(* IEC 61131-3 sources: volt/packages/volt-lsp-iec/test-corpus/pro2193/Device/Plc Logic/Application/01 Main, 4 files *)

(* ---- HardwareButtons.pou ---- *)
{attribute 'global_init_slot' := '50002'}
{attribute 'symbol' := 'none'}
PROGRAM HardwareButtons
VAR_INPUT
	StartCycle			: PushButtonWithObserverFB;
	EndCycle			: PushButtonWithObserverFB;
	Stop				: PushButtonWithObserverFB;
	Reset				: PushButtonWithObserverFB;
	Homing				: PushButtonWithObserverFB;
	F1					: PushButtonFunctionKeyFB;
	F2					: PushButtonFunctionKeyFB;
	{attribute 'symbol' := 'readwrite'}	EnableIML			: PushButtonLedWithHmiFB;
END_VAR
VAR
	startLedTest		: BOOL;
	F1OldObserverCount	: UINT;
	F2OldObserverCount	: UINT;
	speedFooterShow		: BOOL;
	SpeedFooterTimeout	: BTON;
	testestse	: BTON;
	leds				: ARRAY[1..6] OF ILed :=
	[
		StartCycle,
		EndCycle,
		Homing,
		Reset,
		F1,
		F2
	];
	leds2				: ARRAY[1..6] OF ILed :=
	[
		SER.Stacklight.Red,
		SER.Stacklight.Amber,
		SER.Stacklight.Green,
		SER.GateZAxis.ButtonUnLock,
		SER.GateZAxis.ButtonLock,
		ProcessModules.ConveyorControl.ButtonStartNewStack
	];
END_VAR
VAR CONSTANT
	speedFooterShowTime	: REAL	:= 5;	// Show footer for 5 seconds
END_VAR

%LANGUAGE ST
Initialize();

StartCycle(		buttonType		:= enumHWButtons.Start);
EndCycle(		buttonType		:= enumHWButtons.EndCycle);
Stop(			buttonType		:= enumHWButtons.Stop);
Reset(			buttonType		:= enumHWButtons.Reset);
Homing(			buttonType		:= enumHWButtons.Homing);
F1(				buttonType		:= enumHWButtons.F1);
F2(				buttonType		:= enumHWButtons.F2);
EnableIML();
LedTest();

// Switch IML on/off when hardware/software button is pushed
IF EnableIML.ButtonPushed THEN
	PersistentVars.RecipeVars.EnableIML	:= NOT PersistentVars.RecipeVars.EnableIML;
END_IF
IF NOT PersistentVars.RecipeVars.EnableIML THEN
	EnableIML.Off();
ELSIF InjectionMouldingMachine.Data.usiFirstShotsWithoutIML = 0
   OR InjectionMouldingMachine.Unit.ShotCounter > InjectionMouldingMachine.Data.usiFirstShotsWithoutIML
THEN
	EnableIML.SetColors(enumColorList.Lime);
	EnableIML.Solid();
ELSIF SER.OperationMode = SER_OperationModeType.SemiAuto THEN
	EnableIML.SetColors(enumColorList.Lime);
	EnableIML.Solid();
ELSE
	EnableIML.SetColors(enumColorList.Yellow);	// IML temporary disabled during cycle startup
	EnableIML.Solid();
END_IF

IF ErrorHandling.errorActive THEN
	Reset.Flash();
ELSE
	Reset.Off();
END_IF

GlobalVars.Reset S= Reset.ButtonPushed;
GlobalVars.Reset R= Reset.ButtonReleased;

IF F1.ObserverCount <> F1OldObserverCount THEN
	IF F1.ObserverCount > 0 THEN
		F1.Solid();
	ELSE
		F1.Off();
	END_IF
	F1OldObserverCount := F1.ObserverCount;
END_IF

IF F2.ObserverCount <> F2OldObserverCount THEN
	IF F2.ObserverCount > 0 THEN
		F2.Solid();
	ELSE
		F2.Off();
	END_IF
	F2OldObserverCount := F2.ObserverCount;
END_IF

IF SER.InAutomaticOperation
AND SER.OperationMode <> SER_OperationModeType.SemiAuto
THEN
	IF F1.ButtonPushed THEN
		PersistentVars.usiGlobalSERSpeed	:= MAX(5,	PersistentVars.usiGlobalSERSpeed - 5);
		speedFooterShow						:= TRUE;
		HMI.FooterName						:= enumFooterNames.GlobalSpeed;
		SpeedFooterTimeout.Reset();
	END_IF
	IF F2.ButtonPushed THEN
		PersistentVars.usiGlobalSERSpeed	:= MIN(100,	PersistentVars.usiGlobalSERSpeed + 5);
		speedFooterShow						:= TRUE;
		HMI.FooterName						:= enumFooterNames.GlobalSpeed;
		SpeedFooterTimeout.Reset();
	END_IF
END_IF

IF SpeedFooterTimeout.Set(In := speedFooterShow, Pt := speedFooterShowTime) THEN
	speedFooterShow		:= FALSE;
	HMI.FooterName		:= enumFooterNames.None;
END_IF

END_PROGRAM

METHOD PRIVATE Initialize
VAR_INPUT
END_VAR
VAR_INST
	{attribute 'init_on_onlchange'}
	xInitialized	: BOOL;
END_VAR

%LANGUAGE ST
IF xInitialized THEN
	RETURN;
END_IF

startLedTest := TRUE;

xInitialized := TRUE;

END_METHOD

// Do little animation with the leds during startup :)
METHOD PRIVATE LedTest
VAR_INST
	ledTestDuration		: BTON;
	ledTestStep			: BTON;
	i					: INT;
	position			: INT := 1;
END_VAR

%LANGUAGE ST
IF ledTestDuration.Set(In := startLedTest, Pt := 8) THEN
	startLedTest := FALSE;
	position := 1;
	FOR i := 1 TO 6 DO
		leds[i].LedTestStop();
		leds2[i].LedTestStop();
	END_FOR
END_IF

IF ledTestStep.Set(In := startLedTest, Pt := 0.3) THEN
	leds[SEL(position = 1, position - 1, 6)].LedTestOff();
	leds[position].LedTestOn();
	leds[SEL(position = 6, position + 1, 1)].LedTestOn();

	leds2[SEL(position = 1, position - 1, 6)].LedTestOff();
	leds2[position].LedTestOn();

	ledTestStep.Reset();
	Increment.Rollover(input := position, rollover := 6, incrementBy := 1, zeroValue := 1);
END_IF

END_METHOD

(* ---- HMI.pou ---- *)
// By default every variable here has read/write access from the HMI
{attribute 'symbol' := 'readwrite'}
PROGRAM HMI
VAR_INPUT
	xMuteHorn					: BOOL;
	OperationMode				: SER_OperationModeType;	// Unit mode change request from HMI
	FooterName					: enumFooterNames;			// Select active footer type
END_VAR
VAR_OUTPUT
	servoJogMode				: BOOL;						// False: Move to position; True: Servo jogging to sw limit.
	servoJogSpeed				: BOOL;						// False: Slow speed; True: High speed
	UUIDActiveScreen			: STRING(40);
	SemiAutoMode				: enumSemiAutoModeType;		// Choose mode when SER runs in operation mode: Semi-auto
	testMachineWithoutConveyors	: BOOL;						// Disable sensors to testrun the machine without conveyors
	currentUser					: STRING(80);				// Current user
END_VAR
VAR
	ButtonEnableDrives			: PushButtonLedWithHmiFB;
	ButtonEnableMainvalve		: PushButtonLedWithHmiFB;
	ButtonEnableVacuumPumps		: PushButtonLedWithHmiFB;
	ButtonEnableSticker			: PushButtonLedWithHmiFB;
	ButtonEnableCamera			: PushButtonLedWithHmiFB;

	{attribute 'symbol' := 'read'}	SER_State					: PACK_ML.State;
	{attribute 'symbol' := 'read'}	heartbeatToHMI				: UDINT;
	{attribute 'symbol' := 'read'}	ProjectInfo					: ProjectInfoType;
	{attribute 'symbol' := 'read'}	textMessage					: STRING(80);		// Show a custom text message as a popup on the HMI panel.
	{attribute 'symbol' := 'read'}	ipAddressController			: STRING(20);
	{attribute 'symbol' := 'read'}	ipAddressPilz				: STRING(20);
	{attribute 'symbol' := 'read'}	robotSerial					: STRING(7);		// The Serial number of the robot.

	ipAddressEdgePC				: STRING(20)	:= '10.195.0.8';
	communicationPortEdgePC		: UINT			:= 48000;
	heartbeatToPLC				: UDINT;
	logMessageParameterChange	: STRING(255);

	autoLogoffMinutes			: UINT; // Minutes of inactivity after which the current user is being logged off.

	{attribute 'init_on_onlchange'}		// Reset initialized with every online change.
	{attribute 'symbol' := 'none'}	initialized					: BOOL;
	{attribute 'symbol' := 'none'}	startGetControllerIp		: BOOL;
	{attribute 'symbol' := 'none'}	startGetRobotSerial			: BOOL;
	{attribute 'symbol' := 'none'}	heartbeatMissingAlarm		: SetErrorFB();
	{attribute 'symbol' := 'none'}	serialNumberRead			: RobotSerialNumberFB;
END_VAR
VAR CONSTANT
	{attribute 'symbol' := 'none'}	PilzAddToLastOctetOfIp		: BYTE := 2;		// IP address of Pilz PnozMulti will be 2 higher than controller IP. So controller is: 10.100.xxx.10, then Pilz is: : 10.100.xxx.12
END_VAR

%LANGUAGE ST
initialized := initialized OR_ELSE Initialize();

MonitorHeartbeat();

Cyclic();

// Get robot serial number from SD card
serialNumberRead(
	execute				:= startGetRobotSerial,
	controller			:= enumControllerType.C5xxSeries,
	busy				=> ,
	done				=> ,
	errorActive			=> ,
	errorDescription	=> ,
	robotSerial			=> );

IF serialNumberRead.done THEN
	robotSerial				:= serialNumberRead.robotSerial;
	startGetRobotSerial		:= FALSE;
END_IF

END_PROGRAM

// Get the final octet (digit) of an IP address, then increase this digit with another number
METHOD PRIVATE ChangeLastOctetOfIp : STRING(20)
VAR_INPUT
	ipAddress		: STRING(20);
	addTolastOctet	: BYTE;		// number to add to last octet
END_VAR
VAR
	index			: INT;
	lastOctet		: BYTE;
END_VAR

%LANGUAGE ST
index	:= LEN(ipAddress) - 1;	// Get index of last character in string

// Get last index of '.' (ascii: 46)
WHILE ipAddress[index] <> enumASCII.DOT AND index > 0 DO
	index := index - 1;
END_WHILE

IF index > 0 THEN
	lastOctet			:= TO_BYTE(MID(ipAddress, LEN(ipAddress) - 1 - index, index + 2)) + addTolastOctet;
	ChangeLastOctetOfIp := CONCAT(LEFT(ipAddress, index + 1), TO_STRING(lastOctet));
END_IF

END_METHOD

METHOD PRIVATE Cyclic
VAR_INST
	getControllerIp				: GetIPAddressFB;
	UUIDActiveScreenHistory		: ARRAY[0..4] OF STRING(80);
END_VAR
VAR
	i							: USINT;
END_VAR

%LANGUAGE ST
ButtonEnableDrives();
ButtonEnableMainvalve();
ButtonEnableVacuumPumps();
ButtonEnableSticker();
ButtonEnableCamera();

IF SER.xServoDrivesEnabled THEN
	ButtonEnableDrives.SetColors(enumColorList.Lime);
	ButtonEnableDrives.Solid();
ELSIF GlobalVars.EnableServoDrives THEN
	ButtonEnableDrives.SetColors(enumColorList.Blue);
	ButtonEnableDrives.Solid();
ELSE
	ButtonEnableDrives.Off();
END_IF

IF SER.DigIn.xAirPressureOK THEN
	ButtonEnableMainvalve.SetColors(enumColorList.Lime);
	ButtonEnableMainvalve.Solid();
ELSIF GlobalVars.EnableMainvalve THEN
	ButtonEnableMainvalve.SetColors(enumColorList.Blue);
	ButtonEnableMainvalve.Solid();
ELSE
	ButtonEnableMainvalve.Off();
END_IF

IF  SER.VacuumPumps.xVacuumpumpRunning
AND SER.VacuumPumps.xHighVacuumtankFull
AND (SER.VacuumPumps.xLowVacuumtankFull OR SER.VacuumPumps.xOptionDisableVacuumPump2)
THEN
	ButtonEnableVacuumPumps.SetColors(enumColorList.Lime);
	ButtonEnableVacuumPumps.Solid();
ELSIF SER.VacuumPumps.xVacuumpumpRunning THEN
	ButtonEnableVacuumPumps.SetColors(enumColorList.Blue);
	ButtonEnableVacuumPumps.Solid();
ELSE
	ButtonEnableVacuumPumps.SetColors(enumColorList.Gray);
	ButtonEnableVacuumPumps.Off();
END_IF

// Switch IML on/off when software button is pushed
IF ButtonEnableSticker.ButtonPushed AND NOT SER.InAutomaticOperation THEN
	PersistentVars.RecipeVars.EnableSticker	:= NOT PersistentVars.RecipeVars.EnableSticker;
END_IF

ButtonEnableSticker.SetColors(enumColorList.Lime);
IF PersistentVars.RecipeVars.EnableSticker THEN
	ButtonEnableSticker.Solid();
ELSE
	ButtonEnableSticker.Off();
END_IF

// Switch vision system on / off
IF ButtonEnableCamera.ButtonPushed AND NOT SER.InAutomaticOperation THEN			// by customer request only onable/disable camera when machine is off
	PersistentVars.RecipeVars.EnableVision	:= NOT PersistentVars.RecipeVars.EnableVision;
END_IF
ButtonEnableCamera.SetColors(colorOn := enumColorList.Lime);
IF PersistentVars.RecipeVars.EnableVision THEN
	ButtonEnableCamera.Solid();
ELSE
	ButtonEnableCamera.Off();
END_IF

SER_State			:= SER.ActState;

//Get ip addresses of the controller and the Pilz PnozMulti
IF startGetControllerIp THEN
	getControllerIp();
	IF getControllerIp.resultValid THEN
		ipAddressController		:= getControllerIp.currentIp;
		ipAddressPilz			:= ChangeLastOctetOfIp(ipAddressController, PilzAddToLastOctetOfIp);
		startGetControllerIp	:= FALSE;
	END_IF
END_IF

// Debugging: keep a short history of uuids
IF UUIDActiveScreen <> UUIDActiveScreenHistory[0] THEN
	FOR i := 4 TO 1 BY -1 DO
		UUIDActiveScreenHistory[i] := UUIDActiveScreenHistory[i-1];
	END_FOR
	UUIDActiveScreenHistory[0] := UUIDActiveScreen;
END_IF

END_METHOD

// Initializes the FB in the first cycle
METHOD PRIVATE Initialize : BOOL

%LANGUAGE ST
ProjectInfo				:= GetProjectInfo();
startGetControllerIp	:= TRUE;
startGetRobotSerial		:= TRUE;
Initialize				:= TRUE;

END_METHOD

METHOD PRIVATE MonitorHeartbeat
VAR_INST
	heartbeatTimer				: BTON;
	previousHeartbeat			: UDINT;
END_VAR

%LANGUAGE ST
// Send a heartbeat to the HMI every 0,5 sec. (currently not in use)
IF heartbeatTimer.Set(In := TRUE, Pt := 0.5) THEN
	heartbeatTimer.Reset();
	Increment.AnyInt(heartbeatToHMI);
END_IF

// Monitor heartbeat signal from HMI
heartbeatMissingAlarm(
	moduleHandler	:= ErrorHandling.ModuleHandler,
	textRefId		:= General_Unit_Errors,
	errorId			:= 4,		// Missing heartbeat from HMI
	alarmCondition	:= FALSE, //heartbeatToPLC = previousHeartbeat,  // Panel cannot write variables in JS loops..!
	alarmDelay		:= 5.0,
	severity		:= enumErrorSeverity.Warning,
	reaction		:= enumErrorReaction.No_reaction,
	active			=> );

previousHeartbeat := heartbeatToPLC;

// In case of a HMI crash, detach the F1 and F2 buttons from all observers by invalidating the UUID
IF heartbeatMissingAlarm.active THEN
	UUIDActiveScreen := '';
END_IF

END_METHOD

(* ---- HMI_BFU.pou ---- *)
// By default every variable here has read/write access from the HMI
{attribute 'symbol' := 'readwrite'}
// Handle the BFU specific buttons
PROGRAM HMI_BFU
VAR_INPUT
	OperationMode				: SER_OperationModeType;	// Unit mode change request from HMI
END_VAR
VAR_OUTPUT
	UUIDActiveScreen			: STRING(40);
END_VAR
VAR
	ButtonEnableDrives			: PushButtonLedWithHmiFB;
	ButtonEnableMainvalve		: PushButtonLedWithHmiFB;
	ButtonEnableVacuumPumps		: PushButtonLedWithHmiFB;

	{attribute 'symbol' := 'read'}	BFU_State					: PACK_ML.State;
END_VAR

%LANGUAGE ST
Initialize();

ButtonEnableDrives();
ButtonEnableMainvalve();
ButtonEnableVacuumPumps();

IF BFU.xServoDrivesEnabled THEN
	ButtonEnableDrives.SetColors(enumColorList.Lime);
	ButtonEnableDrives.Solid();
ELSIF GlobalVars_BFU.EnableServoDrives THEN
	ButtonEnableDrives.SetColors(enumColorList.Blue);
	ButtonEnableDrives.Solid();
ELSE
	ButtonEnableDrives.Off();
END_IF

IF BFU.DigIn.xAirPressureOK THEN
	ButtonEnableMainvalve.SetColors(enumColorList.Lime);
	ButtonEnableMainvalve.Solid();
ELSIF GlobalVars_BFU.EnableMainvalve THEN
	ButtonEnableMainvalve.SetColors(enumColorList.Blue);
	ButtonEnableMainvalve.Solid();
ELSE
	ButtonEnableMainvalve.Off();
END_IF

BFU_State			:= BFU.ActState;

END_PROGRAM

METHOD PRIVATE Initialize
VAR_INPUT
END_VAR
VAR_INST
	xInitialized	: BOOL;
END_VAR

%LANGUAGE ST
IF xInitialized THEN
	RETURN;
END_IF

xInitialized := TRUE;

END_METHOD

(* ---- Main.pou ---- *)
PROGRAM Main
VAR
	StartupTimer	: BTON;
	taskInfo				: CmpIecTask.Task_Info2;
END_VAR

%LANGUAGE ST
__TRY
taskInfo	:= TaskGetInfo();
IF NOT StartupTimer.Set(TRUE, 1) THEN	// Delay before starting program. The first PLC cycle the I/Q is not updated yet.
	IQ_Handling();
	RETURN;
END_IF

__CATCH(GVL_Exceptions.aeExceptionCodes[eExceptionCodes.MainTask])
	GVL_Exceptions.xException := TRUE;
	GVL_Exceptions.iCounter := GVL_Exceptions.iCounter + 1;
__ENDTRY

__TRY TimeSettings();		__CATCH(GVL_Exceptions.aeExceptionCodes[eExceptionCodes.TimeSettings])	GVL_Exceptions.xException := TRUE;	GVL_Exceptions.iCounter := GVL_Exceptions.iCounter + 1;		__ENDTRY		// Get or set the current date / time
__TRY EtherCAT_Diag();		__CATCH(GVL_Exceptions.aeExceptionCodes[eExceptionCodes.EtherCAT_Diag])	GVL_Exceptions.xException := TRUE;	GVL_Exceptions.iCounter := GVL_Exceptions.iCounter + 1;		__ENDTRY	// Get diagnostics about the EtherCAT connection
__TRY ErrorHandling();		__CATCH(GVL_Exceptions.aeExceptionCodes[eExceptionCodes.ErrorHandling])	GVL_Exceptions.xException := TRUE;	GVL_Exceptions.iCounter := GVL_Exceptions.iCounter + 1;		__ENDTRY
__TRY HardwareButtons();	__CATCH(GVL_Exceptions.aeExceptionCodes[eExceptionCodes.HardwareButtons])	GVL_Exceptions.xException := TRUE;	GVL_Exceptions.iCounter := GVL_Exceptions.iCounter + 1;		__ENDTRY
__TRY BfuButtons();			__CATCH(GVL_Exceptions.aeExceptionCodes[eExceptionCodes.BfuButtons])	GVL_Exceptions.xException := TRUE;	GVL_Exceptions.iCounter := GVL_Exceptions.iCounter + 1;		__ENDTRY
__TRY HMI();				__CATCH(GVL_Exceptions.aeExceptionCodes[eExceptionCodes.HMI])	GVL_Exceptions.xException := TRUE;	GVL_Exceptions.iCounter := GVL_Exceptions.iCounter + 1;		__ENDTRY		// Setup communication with HMI panel
__TRY HMI_BFU();			__CATCH(GVL_Exceptions.aeExceptionCodes[eExceptionCodes.HMI_BFU])	GVL_Exceptions.xException := TRUE;	GVL_Exceptions.iCounter := GVL_Exceptions.iCounter + 1;		__ENDTRY
__TRY HardwareUnits();		__CATCH(GVL_Exceptions.aeExceptionCodes[eExceptionCodes.HardwareUnits])	GVL_Exceptions.xException := TRUE;	GVL_Exceptions.iCounter := GVL_Exceptions.iCounter + 1;		__ENDTRY	// First initialize hardware units (lowest level)
__TRY ProcessModules();		__CATCH(GVL_Exceptions.aeExceptionCodes[eExceptionCodes.ProcessModules])	GVL_Exceptions.xException := TRUE;	GVL_Exceptions.iCounter := GVL_Exceptions.iCounter + 1;		__ENDTRY	// Then initialize process units
__TRY SER();				__CATCH(GVL_Exceptions.aeExceptionCodes[eExceptionCodes.SER])	GVL_Exceptions.xException := TRUE;	GVL_Exceptions.iCounter := GVL_Exceptions.iCounter + 1;		__ENDTRY		// SER need to be last in the list, so all in_out variables are connected
__TRY BFU();				__CATCH(GVL_Exceptions.aeExceptionCodes[eExceptionCodes.BFU])	GVL_Exceptions.xException := TRUE;	GVL_Exceptions.iCounter := GVL_Exceptions.iCounter + 1;		__ENDTRY		// BFU need to be last in the list, so all in_out variables are connected
__TRY IQ_Handling();		__CATCH(GVL_Exceptions.aeExceptionCodes[eExceptionCodes.IQ_Handling])	GVL_Exceptions.xException := TRUE;	GVL_Exceptions.iCounter := GVL_Exceptions.iCounter + 1;		__ENDTRY		// Read and write all I/Q slices

END_PROGRAM
